// Mitsubishi GX Works2 project: 랜덤 타이머   PLC: Q02/Q02H

PROGRAM MAIN
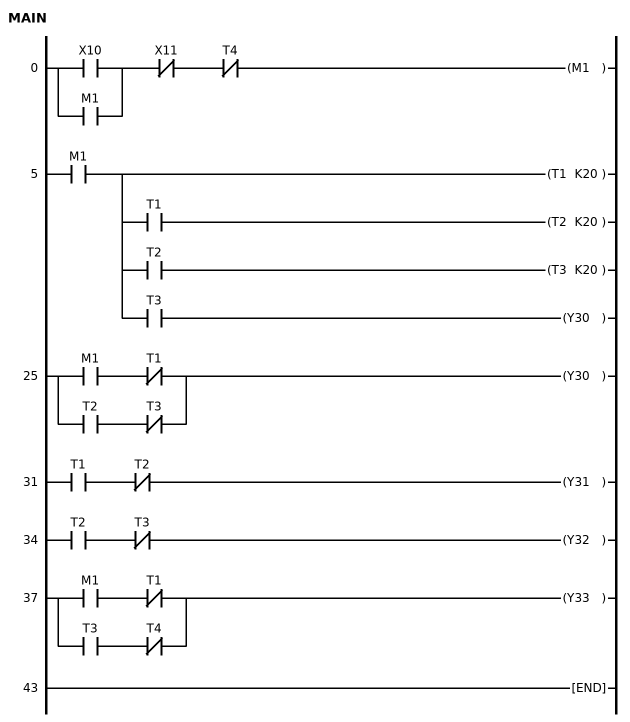
0     LD      X10
      OR      M1
      ANI     X11
      ANI     T4
      OUT     M1
5     LD      M1
      OUT     T1 K20
      MPS
      AND     T1
      OUT     T2 K20
      MRD
      AND     T2
      OUT     T3 K20
      MPP
      AND     T3
      OUT     Y30
25    LD      M1
      ANI     T1
      LD      T2
      ANI     T3
      ORB
      OUT     Y30
31    LD      T1
      ANI     T2
      OUT     Y31
34    LD      T2
      ANI     T3
      OUT     Y32
37    LD      M1
      ANI     T1
      LD      T3
      ANI     T4
      ORB
      OUT     Y33
43    END
END_PROGRAM
